(* IEC 61131-3 sources: SIMATIC-AX-Workshop-NL/src, 2 files *)

(* ---- library.st ---- *)
NAMESPACE MotorLibrary

    CLASS PUBLIC Motor
        VAR PRIVATE
            _started : BOOL;
        END_VAR

        VAR PRIVATE

        END_VAR

        METHOD PUBLIC Start : BOOL
            _started := FALSE;
            Start := TRUE;
        END_METHOD
    END_CLASS

END_NAMESPACE

(* ---- wrapper.st ---- *)
NAMESPACE MotorLibrary

    FUNCTION_BLOCK MotorWrapper
        VAR_INPUT
            start : BOOL;
        END_VAR
        VAR
            m : Motor;
        END_VAR

        IF start THEN
            m.Start();
        END_IF;
    END_FUNCTION_BLOCK

END_NAMESPACE
